TYPE BeaconItem :
STRUCT
	Number : INT;
	Clock : Clock;
	Output : REFERENCE TO BOOL;
	Duration : TON;
	DurationTime : TIME;
END_STRUCT
END_TYPE

(* stored: Version 1.1.0.1
   DUT BeaconItem: Id {e4887bfd-7446-0050-2144-2d137e0b82fe} *)
